FUNCTION WConcat7 : WSTRING(255)
VAR_INPUT
	wsExpression1: WSTRING(255);
	wsExpression2: WSTRING(255);
	wsExpression3: WSTRING(255);
	wsExpression4: WSTRING(255);
	wsExpression5: WSTRING(255);
	wsExpression6: WSTRING(255);
	wsExpression7: WSTRING(255);
END_VAR

WConcat7 := WCONCAT(wsExpression1, wsExpression2);
WConcat7 := WCONCAT(WConcat7, wsExpression3);
WConcat7 := WCONCAT(WConcat7, wsExpression4);
WConcat7 := WCONCAT(WConcat7, wsExpression5);
WConcat7 := WCONCAT(WConcat7, wsExpression6);
WConcat7 := WCONCAT(WConcat7, wsExpression7);

END_FUNCTION

(* stored: Version 1.1.0.1, ProductVersion 3.1.4024.11
   POU WConcat7: Id {04183ee3-41f1-4c17-93b4-c746f0078895}, SpecialFunc None *)
